FUNCTION TryConvert_DINT_TO_INT : BOOL
VAR_INPUT
	in : DINT;
	out : REFERENCE TO INT;
END_VAR

IF in > DatatypeLimits.MAX_VALUE_OF_DINT_WHICH_CAN_BE_HELD_IN_A_INT THEN
	RETURN;
END_IF

IF in < DatatypeLimits.MIN_VALUE_OF_DINT_WHICH_CAN_BE_HELD_IN_A_INT THEN
	RETURN;
END_IF

out := DINT_TO_INT(in);
TryConvert_DINT_TO_INT := TRUE;

END_FUNCTION

(* stored: Version 1.1.0.1, ProductVersion 3.1.4024.12
   POU TryConvert_DINT_TO_INT: Id {d10a9427-91b5-435b-b012-3d31a2685e72}, SpecialFunc None *)
